// TIA Portal V17 export
// export: Created 2021-12-03T08:13:03.045766Z, ExportSetting WithDefaults, DisplayName Totally Integrated Automation Portal, DisplayVersion V17, DisplayName TIA Portal Openness, DisplayVersion V17, DisplayName TIA Portal Version Control Interface, DisplayVersion V17, DisplayName STEP 7 Professional, DisplayVersion V17, DisplayName STEP 7 Safety, DisplayVersion V17, DisplayName WinCC Advanced, DisplayVersion V17
FUNCTION "FC_AcceleratorCtrl" : Void   // FC62, FBD
VERSION : 0.1
// stored: AutoNumber false, IsIECCheckEnabled false, UDAEnableTagReadback false
   VAR_TEMP
      T_Acc_RstSig : Bool;
      T_WarmUpSig : Bool;
      T_FullWarmUpSig : Bool;
      T_NoEStp : Bool;   // Сигнал аварийного останова
      T_ChDose : Bool;
      T_RFOnRq : Bool;   // Запрос на включение СВЧ
      T_RF_On : Bool;   // Включить СВЧ
      T_XRayOnRq : Bool;   // Запрос на включение ТИ
      T_XRay_On : Bool;   // ТИ включить
      Mod400V_Fb : Bool;
      AccMod220V_Fb : Bool;
      Mod380V_PwrOnRq : Bool;
      Mod380V_PwrOffRq : Bool;
      T_AccFlt : Bool;
   END_VAR
BEGIN

REGION Network 2: Режим измененной дозы
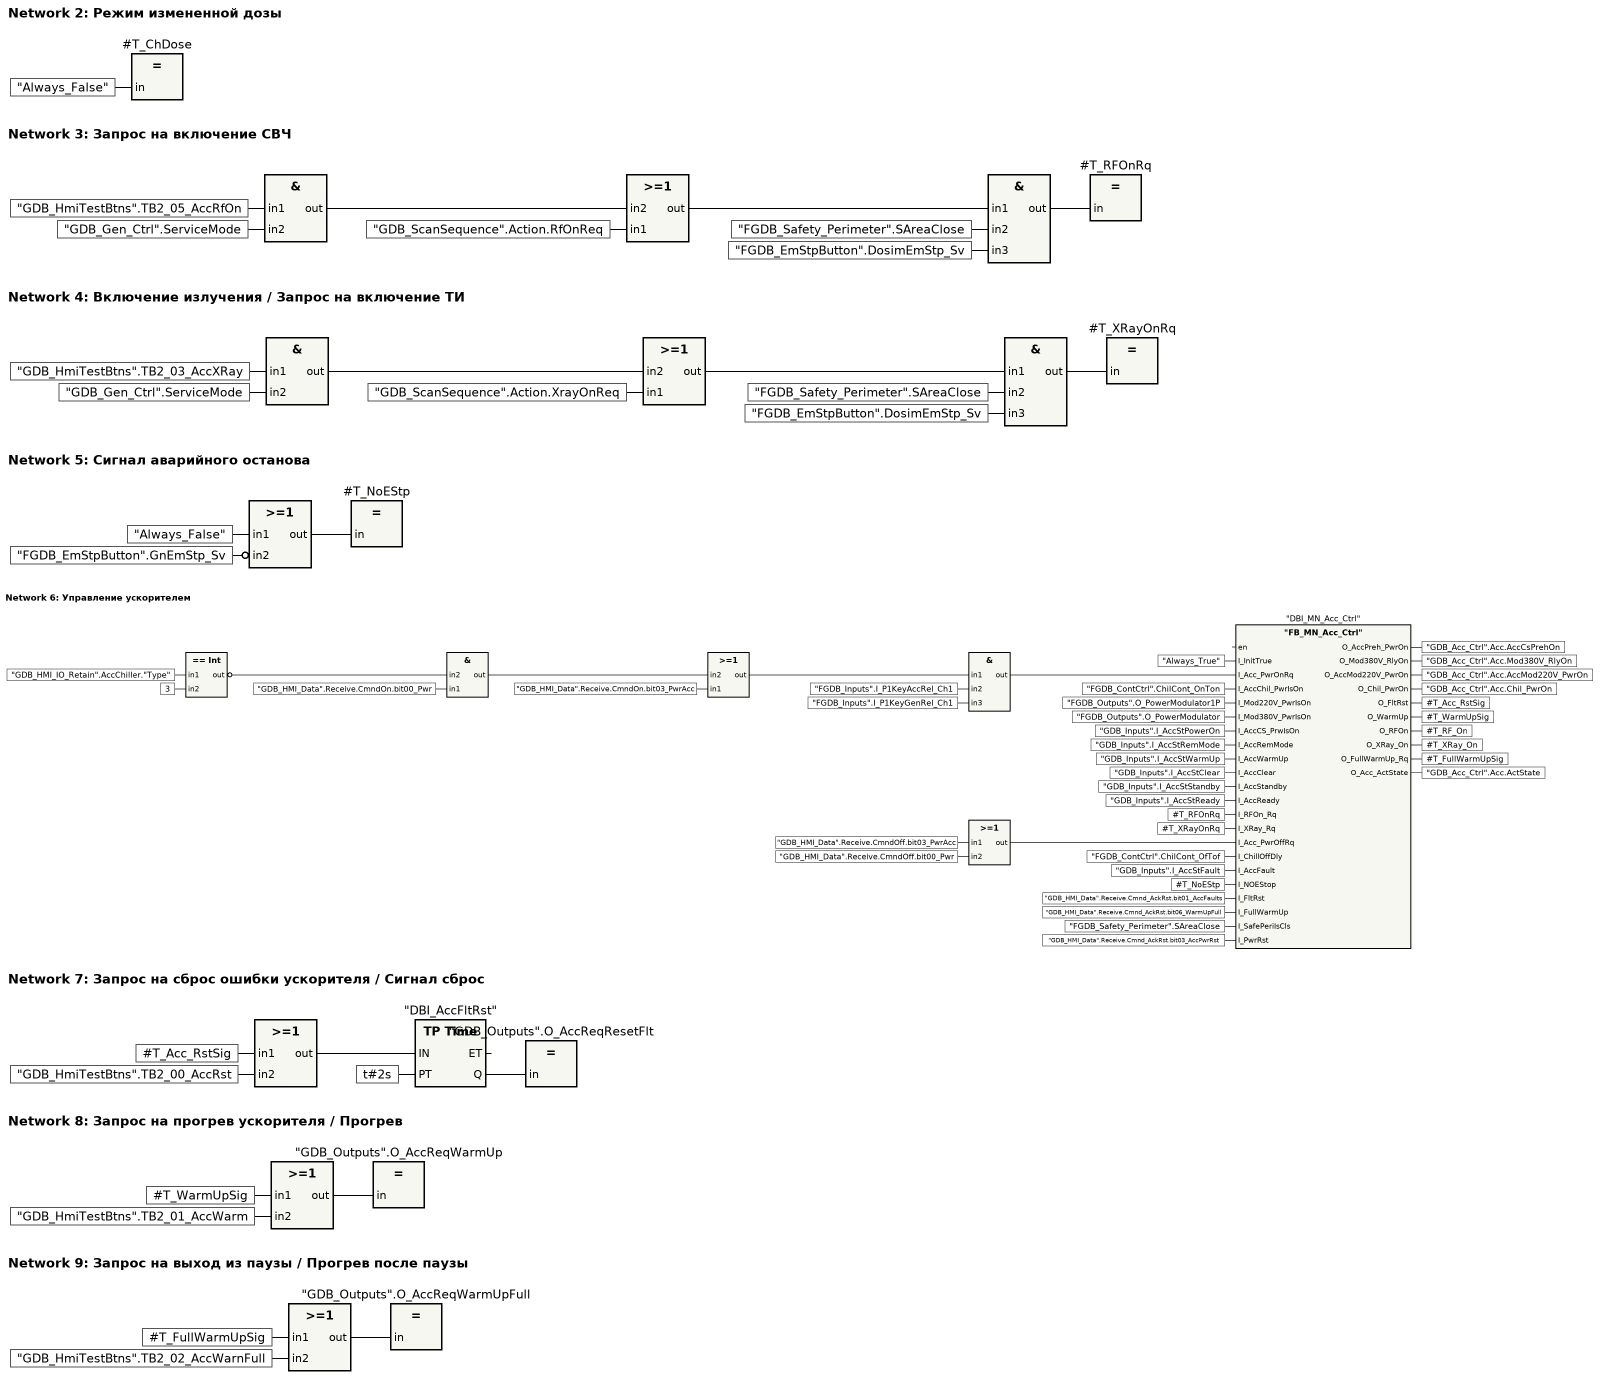
   #T_ChDose := "Always_False";
END_REGION

REGION Network 3: Запрос на включение СВЧ
   #T_RFOnRq := (("GDB_HmiTestBtns".TB2_05_AccRfOn AND "GDB_Gen_Ctrl".ServiceMode) OR "GDB_ScanSequence".Action.RfOnReq) AND "FGDB_Safety_Perimeter".SAreaClose AND "FGDB_EmStpButton".DosimEmStp_Sv;
END_REGION

REGION Network 4: Включение излучения / Запрос на включение ТИ
   #T_XRayOnRq := (("GDB_HmiTestBtns".TB2_03_AccXRay AND "GDB_Gen_Ctrl".ServiceMode) OR "GDB_ScanSequence".Action.XrayOnReq) AND "FGDB_Safety_Perimeter".SAreaClose AND "FGDB_EmStpButton".DosimEmStp_Sv;
END_REGION

REGION Network 5: Сигнал аварийного останова
   #T_NoEStp := "Always_False" OR NOT "FGDB_EmStpButton".GnEmStp_Sv;
END_REGION

REGION Network 6: Управление ускорителем
   "DBI_MN_Acc_Ctrl"(I_InitTrue := "Always_True",   // "FB_MN_Acc_Ctrl"
                     I_Acc_PwrOnRq := ((NOT ("GDB_HMI_IO_Retain".AccChiller."Type" = 3) AND "GDB_HMI_Data".Receive.CmndOn.bit00_Pwr) OR "GDB_HMI_Data".Receive.CmndOn.bit03_PwrAcc) AND "FGDB_Inputs".I_P1KeyAccRel_Ch1 AND "FGDB_Inputs".I_P1KeyGenRel_Ch1,
                     I_AccChil_PwrIsOn := "FGDB_ContCtrl".ChilCont_OnTon,
                     I_Mod220V_PwrIsOn := "FGDB_Outputs".O_PowerModulator1P,
                     I_Mod380V_PwrIsOn := "FGDB_Outputs".O_PowerModulator,
                     I_AccCS_PrwIsOn := "GDB_Inputs".I_AccStPowerOn,
                     I_AccRemMode := "GDB_Inputs".I_AccStRemMode,
                     I_AccWarmUp := "GDB_Inputs".I_AccStWarmUp,
                     I_AccClear := "GDB_Inputs".I_AccStClear,
                     I_AccStandby := "GDB_Inputs".I_AccStStandby,
                     I_AccReady := "GDB_Inputs".I_AccStReady,
                     I_RFOn_Rq := #T_RFOnRq,
                     I_XRay_Rq := #T_XRayOnRq,
                     I_Acc_PwrOffRq := "GDB_HMI_Data".Receive.CmndOff.bit03_PwrAcc OR "GDB_HMI_Data".Receive.CmndOff.bit00_Pwr,
                     I_ChillOffDly := "FGDB_ContCtrl".ChilCont_OfTof,
                     I_AccFault := "GDB_Inputs".I_AccStFault,
                     I_NOEStop := #T_NoEStp,
                     I_FltRst := "GDB_HMI_Data".Receive.Cmnd_AckRst.bit01_AccFaults,
                     I_FullWarmUp := "GDB_HMI_Data".Receive.Cmnd_AckRst.bit06_WarmUpFull,
                     I_SafePeriIsCls := "FGDB_Safety_Perimeter".SAreaClose,
                     I_PwrRst := "GDB_HMI_Data".Receive.Cmnd_AckRst.bit03_AccPwrRst,
                     O_AccPreh_PwrOn => "GDB_Acc_Ctrl".Acc.AccCsPrehOn,
                     O_Mod380V_RlyOn => "GDB_Acc_Ctrl".Acc.Mod380V_RlyOn,
                     O_AccMod220V_PwrOn => "GDB_Acc_Ctrl".Acc.AccMod220V_PwrOn,
                     O_Chil_PwrOn => "GDB_Acc_Ctrl".Acc.Chil_PwrOn,
                     O_FltRst => #T_Acc_RstSig,
                     O_WarmUp => #T_WarmUpSig,
                     O_RFOn => #T_RF_On,
                     O_XRay_On => #T_XRay_On,
                     O_FullWarmUp_Rq => #T_FullWarmUpSig,
                     O_Acc_ActState => "GDB_Acc_Ctrl".Acc.ActState);
END_REGION

REGION Network 7: Запрос на сброс ошибки ускорителя / Сигнал сброс
   "DBI_AccFltRst".TP(IN := #T_Acc_RstSig OR "GDB_HmiTestBtns".TB2_00_AccRst, PT := t#2s);
   "GDB_Outputs".O_AccReqResetFlt := "DBI_AccFltRst".Q;
END_REGION

REGION Network 8: Запрос на прогрев ускорителя / Прогрев
   "GDB_Outputs".O_AccReqWarmUp := #T_WarmUpSig OR "GDB_HmiTestBtns".TB2_01_AccWarm;
END_REGION

REGION Network 9: Запрос на выход из паузы / Прогрев после паузы
   "GDB_Outputs".O_AccReqWarmUpFull := #T_FullWarmUpSig OR "GDB_HmiTestBtns".TB2_02_AccWarnFull;
END_REGION

REGION Network 10: Запрос на изменение дозы
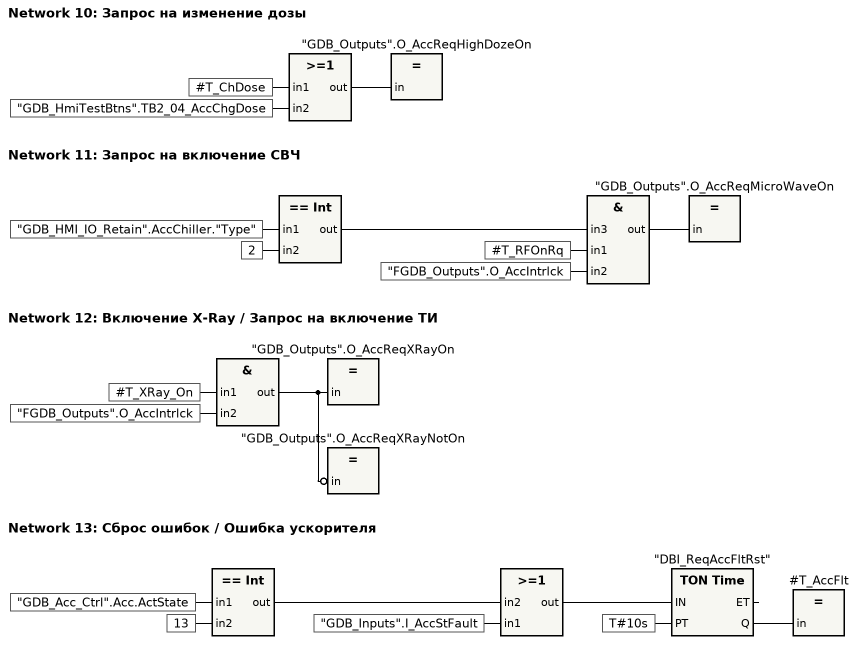
   "GDB_Outputs".O_AccReqHighDozeOn := #T_ChDose OR "GDB_HmiTestBtns".TB2_04_AccChgDose;
END_REGION

REGION Network 11: Запрос на включение СВЧ
   "GDB_Outputs".O_AccReqMicroWaveOn := ("GDB_HMI_IO_Retain".AccChiller."Type" = 2) AND #T_RFOnRq AND "FGDB_Outputs".O_AccIntrlck;
END_REGION

REGION Network 12: Включение X-Ray / Запрос на включение ТИ
   "GDB_Outputs".O_AccReqXRayOn := #T_XRay_On AND "FGDB_Outputs".O_AccIntrlck;
   "GDB_Outputs".O_AccReqXRayNotOn := NOT "GDB_Outputs".O_AccReqXRayOn;
END_REGION

REGION Network 13: Сброс ошибок / Ошибка ускорителя
   "DBI_ReqAccFltRst".TON(IN := ("GDB_Acc_Ctrl".Acc.ActState = 13) OR "GDB_Inputs".I_AccStFault, PT := T#10s);
   #T_AccFlt := "DBI_ReqAccFltRst".Q;
END_REGION
END_FUNCTION
